// TIA Portal V18 export
// export: Created 2025-12-01T12:38:34.6445112Z, ExportSetting None, DisplayName Totally Integrated Automation Portal, DisplayVersion V18 Update 5, DisplayName TIA Portal Openness, DisplayVersion V18 Update 5, DisplayName TIA Portal Teamcenter Gateway, DisplayVersion V18, DisplayName TIA Portal Version Control Interface, DisplayVersion V18, DisplayName STEP 7 Professional, DisplayVersion V18 Update 5, DisplayName STEP 7 Safety, DisplayVersion V18, DisplayName WinCC Professional, DisplayVersion V18 Update 5
FUNCTION_BLOCK "ST10_Stopper_FB"   // FB1160, LAD
{ S7_Optimized_Access := 'TRUE' }
// stored: AutoNumber false, MemoryReserve 100, SetENOAutomatically false
   VAR
      FB_Stopper_Instance { S7_SetPoint := 'True'} : Array[1..3] of "FB_Stopper";
   END_VAR
BEGIN

REGION Network 1 (SCL): A-托盘缓存阻挡气缸
       (*  
       REGION 允许释放条件,根据实际完善
           //马达运行中且工位一允许进料
           IF "ST350_Motor_InterfaceDB".aDev[1].Run  THEN
               "ST350_Stopper_InterfaceDB".Command[1].In.iReleaseClear := TRUE;
           ELSE
               "ST350_Stopper_InterfaceDB".Command[1].In.iReleaseClear := FALSE;
           END_IF;
       END_REGION

       REGION IO_image
           //InPut
           "ST350_Stopper_InterfaceDB".Command[1].In.iSensor := "iBurfferPalletDetection";//本站托盘到位
           "ST350_Stopper_InterfaceDB".Command[1].In.iNextSensor := "iWork01PalletDetection";//后站托盘到位
           "ST350_Stopper_InterfaceDB".Command[1].In.iNextValve := "oA-Lifting-01StopperCylinder";//后站挡停输出

           // //OutPut
            "ST10Cylinder".Cy[5].Inout.AutoGoWork:= "ST350_Stopper_InterfaceDB".Command[1].Out.oValve;//本站挡停输出
       END_REGION


       *)
END_REGION

REGION Network 2: #FB_Stopper_Instance[1] A-托盘缓存阻挡气缸
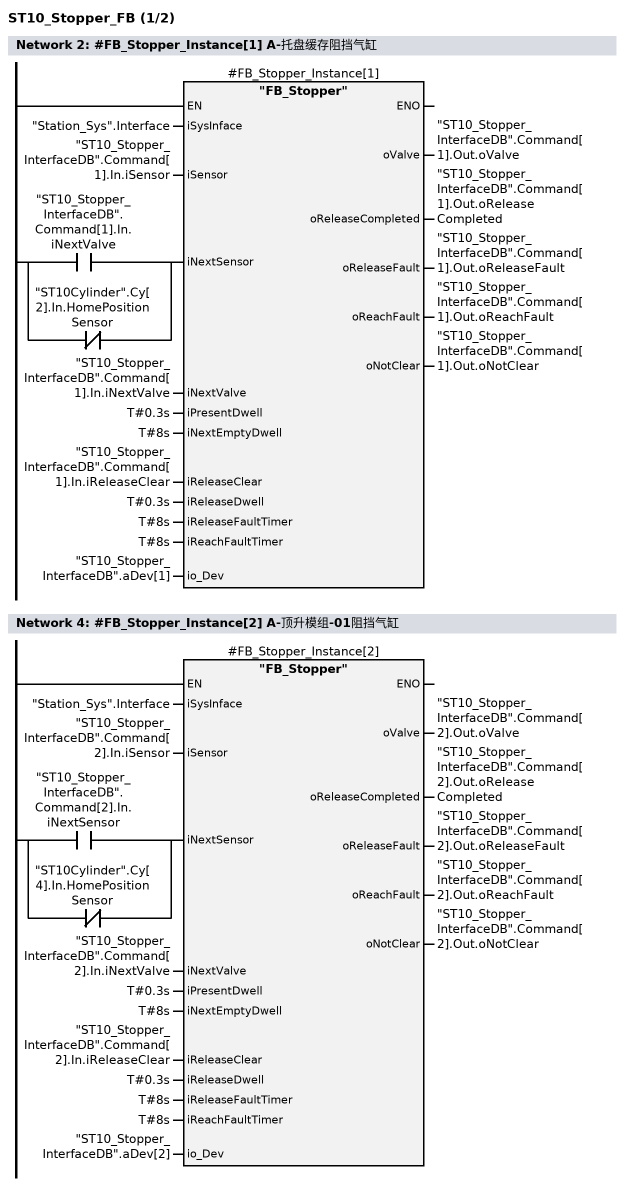
   RUNG wire#powerrail
      #FB_Stopper_Instance[1](iNextSensor := wire#w1, iSysInface := "Station_Sys".Interface, iSensor := "ST10_Stopper_InterfaceDB".Command[1].In.iSensor, iNextValve := "ST10_Stopper_InterfaceDB".Command[1].In.iNextValve, iPresentDwell := T#0.3s, iNextEmptyDwell := T#8s, iReleaseClear := "ST10_Stopper_InterfaceDB".Command[1].In.iReleaseClear, iReleaseDwell := T#0.3s, iReleaseFaultTimer := T#8s, iReachFaultTimer := T#8s, io_Dev := "ST10_Stopper_InterfaceDB".aDev[1], oValve => "ST10_Stopper_InterfaceDB".Command[1].Out.oValve, oReleaseCompleted => "ST10_Stopper_InterfaceDB".Command[1].Out.oReleaseCompleted, oReleaseFault => "ST10_Stopper_InterfaceDB".Command[1].Out.oReleaseFault, oReachFault => "ST10_Stopper_InterfaceDB".Command[1].Out.oReachFault, oNotClear => "ST10_Stopper_InterfaceDB".Command[1].Out.oNotClear)
   END_RUNG
   RUNG wire#powerrail
      Contact( "ST10_Stopper_InterfaceDB".Command[1].In.iNextValve )
   END_RUNG wire#w1
   RUNG wire#powerrail
      I_Contact( "ST10Cylinder".Cy[2].In.HomePositionSensor )
   END_RUNG wire#w1
   // the same network as SCL:
   #FB_Stopper_Instance[1](iSysInface := "Station_Sys".Interface,   // "FB_Stopper"
                           iSensor := "ST10_Stopper_InterfaceDB".Command[1].In.iSensor,
                           iNextSensor := "ST10_Stopper_InterfaceDB".Command[1].In.iNextValve OR NOT "ST10Cylinder".Cy[2].In.HomePositionSensor,
                           iNextValve := "ST10_Stopper_InterfaceDB".Command[1].In.iNextValve,
                           iPresentDwell := T#0.3s,
                           iNextEmptyDwell := T#8s,
                           iReleaseClear := "ST10_Stopper_InterfaceDB".Command[1].In.iReleaseClear,
                           iReleaseDwell := T#0.3s,
                           iReleaseFaultTimer := T#8s,
                           iReachFaultTimer := T#8s,
                           io_Dev := "ST10_Stopper_InterfaceDB".aDev[1],
                           oValve => "ST10_Stopper_InterfaceDB".Command[1].Out.oValve,
                           oReleaseCompleted => "ST10_Stopper_InterfaceDB".Command[1].Out.oReleaseCompleted,
                           oReleaseFault => "ST10_Stopper_InterfaceDB".Command[1].Out.oReleaseFault,
                           oReachFault => "ST10_Stopper_InterfaceDB".Command[1].Out.oReachFault,
                           oNotClear => "ST10_Stopper_InterfaceDB".Command[1].Out.oNotClear);
END_REGION

REGION Network 3 (SCL): A-顶升模组-01阻挡气缸
   (*
   REGION 允许释放条件,根据实际完善:顶升下降且线体运行中
       IF "ST10Cylinder".Cy[2].In.HomePositionSensor AND ("ST350_Motor_InterfaceDB".aDev[1].Run OR "Station_Sys".Manual.Mode) THEN//
           "ST350_Stopper_InterfaceDB".Command[2].In.iReleaseClear := True;
       ELSE
           "ST350_Stopper_InterfaceDB".Command[2].In.iReleaseClear := FALSE;
       END_IF;
   END_REGION

   REGION IO_image
       //InPut
       "ST350_Stopper_InterfaceDB".Command[2].In.iSensor := "iWork01PalletDetection";//本站托盘到位
       "ST350_Stopper_InterfaceDB".Command[2].In.iNextSensor := "iWork02PalletDetection";//后站托盘到位
       "ST350_Stopper_InterfaceDB".Command[2].In.iNextValve := "oA-Lifting-02StopperCylinder";//后站挡停输出

       // //OutPut
        "ST10Cylinder".Cy[1].Inout.AutoGoWork:= "ST350_Stopper_InterfaceDB".Command[2].Out.oValve;//本站挡停输出
   END_REGION

   *0
END_REGION

REGION Network 4: #FB_Stopper_Instance[2] A-顶升模组-01阻挡气缸
   RUNG wire#powerrail
      #FB_Stopper_Instance[2](iNextSensor := wire#w1, iSysInface := "Station_Sys".Interface, iSensor := "ST10_Stopper_InterfaceDB".Command[2].In.iSensor, iNextValve := "ST10_Stopper_InterfaceDB".Command[2].In.iNextValve, iPresentDwell := T#0.3s, iNextEmptyDwell := T#8s, iReleaseClear := "ST10_Stopper_InterfaceDB".Command[2].In.iReleaseClear, iReleaseDwell := T#0.3s, iReleaseFaultTimer := T#8s, iReachFaultTimer := T#8s, io_Dev := "ST10_Stopper_InterfaceDB".aDev[2], oValve => "ST10_Stopper_InterfaceDB".Command[2].Out.oValve, oReleaseCompleted => "ST10_Stopper_InterfaceDB".Command[2].Out.oReleaseCompleted, oReleaseFault => "ST10_Stopper_InterfaceDB".Command[2].Out.oReleaseFault, oReachFault => "ST10_Stopper_InterfaceDB".Command[2].Out.oReachFault, oNotClear => "ST10_Stopper_InterfaceDB".Command[2].Out.oNotClear)
   END_RUNG
   RUNG wire#powerrail
      Contact( "ST10_Stopper_InterfaceDB".Command[2].In.iNextSensor )
   END_RUNG wire#w1
   RUNG wire#powerrail
      I_Contact( "ST10Cylinder".Cy[4].In.HomePositionSensor )
   END_RUNG wire#w1
   // the same network as SCL:
   #FB_Stopper_Instance[2](iSysInface := "Station_Sys".Interface,   // "FB_Stopper"
                           iSensor := "ST10_Stopper_InterfaceDB".Command[2].In.iSensor,
                           iNextSensor := "ST10_Stopper_InterfaceDB".Command[2].In.iNextSensor OR NOT "ST10Cylinder".Cy[4].In.HomePositionSensor,
                           iNextValve := "ST10_Stopper_InterfaceDB".Command[2].In.iNextValve,
                           iPresentDwell := T#0.3s,
                           iNextEmptyDwell := T#8s,
                           iReleaseClear := "ST10_Stopper_InterfaceDB".Command[2].In.iReleaseClear,
                           iReleaseDwell := T#0.3s,
                           iReleaseFaultTimer := T#8s,
                           iReachFaultTimer := T#8s,
                           io_Dev := "ST10_Stopper_InterfaceDB".aDev[2],
                           oValve => "ST10_Stopper_InterfaceDB".Command[2].Out.oValve,
                           oReleaseCompleted => "ST10_Stopper_InterfaceDB".Command[2].Out.oReleaseCompleted,
                           oReleaseFault => "ST10_Stopper_InterfaceDB".Command[2].Out.oReleaseFault,
                           oReachFault => "ST10_Stopper_InterfaceDB".Command[2].Out.oReachFault,
                           oNotClear => "ST10_Stopper_InterfaceDB".Command[2].Out.oNotClear);
END_REGION

REGION Network 5 (SCL): A-顶升模组-02阻挡气缸
   //允许释放条件,根据实际完善:顶升下降且线体运行中
   (*

   REGION IOimage
       //InPut
       "ST350_Stopper_InterfaceDB".Command[3].In.iSensor := "iWork02PalletDetection";//本站托盘到位
       "ST350_Stopper_InterfaceDB".Command[3].In.iNextSensor := "iD-LiftingDetection" AND NOT "iD-LiftingINDetection" ;//后站托盘到位

       //替换后站挡停释放信号：升降机在下&顶升下&无料&允许金托盘
       // "ST350_Stopper_InterfaceDB".Command[3].In.iNextValve := ;//后站挡停输出

       // //OutPut
        "ST10Cylinder".Cy[3].Inout.AutoGoWork := "ST350_Stopper_InterfaceDB".Command[3].Out.oValve;//本站挡停输出


   END_REGION

   *)
END_REGION

REGION Network 6: #FB_Stopper_Instance[3] A-顶升模组-02阻挡气缸
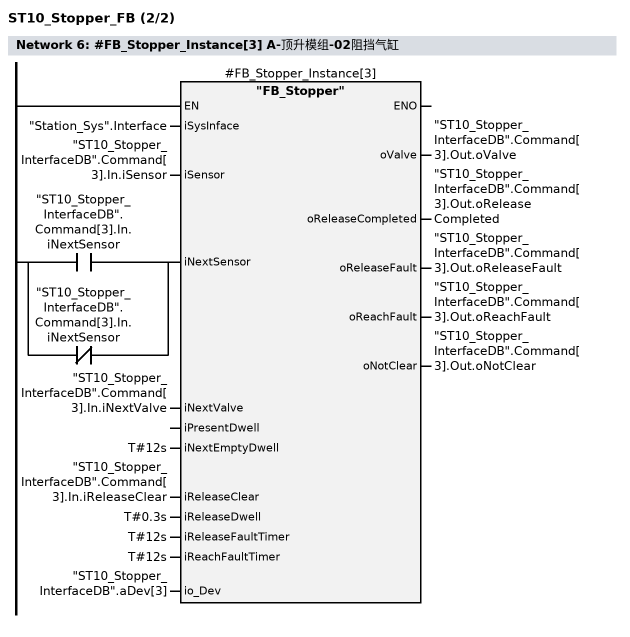
   RUNG wire#powerrail
      #FB_Stopper_Instance[3](iNextSensor := wire#w1, iSysInface := "Station_Sys".Interface, iSensor := "ST10_Stopper_InterfaceDB".Command[3].In.iSensor, iNextValve := "ST10_Stopper_InterfaceDB".Command[3].In.iNextValve, iPresentDwell :=, iNextEmptyDwell := T#12s, iReleaseClear := "ST10_Stopper_InterfaceDB".Command[3].In.iReleaseClear, iReleaseDwell := T#0.3s, iReleaseFaultTimer := T#12s, iReachFaultTimer := T#12s, io_Dev := "ST10_Stopper_InterfaceDB".aDev[3], oValve => "ST10_Stopper_InterfaceDB".Command[3].Out.oValve, oReleaseCompleted => "ST10_Stopper_InterfaceDB".Command[3].Out.oReleaseCompleted, oReleaseFault => "ST10_Stopper_InterfaceDB".Command[3].Out.oReleaseFault, oReachFault => "ST10_Stopper_InterfaceDB".Command[3].Out.oReachFault, oNotClear => "ST10_Stopper_InterfaceDB".Command[3].Out.oNotClear)
   END_RUNG
   RUNG wire#powerrail
      Contact( "ST10_Stopper_InterfaceDB".Command[3].In.iNextSensor )
   END_RUNG wire#w1
   RUNG wire#powerrail
      I_Contact( "ST10_Stopper_InterfaceDB".Command[3].In.iNextSensor )
   END_RUNG wire#w1
   // the same network as SCL:
   #FB_Stopper_Instance[3](iSysInface := "Station_Sys".Interface,   // "FB_Stopper"
                           iSensor := "ST10_Stopper_InterfaceDB".Command[3].In.iSensor,
                           iNextSensor := "ST10_Stopper_InterfaceDB".Command[3].In.iNextSensor OR NOT "ST10_Stopper_InterfaceDB".Command[3].In.iNextSensor,
                           iNextValve := "ST10_Stopper_InterfaceDB".Command[3].In.iNextValve,
                           iNextEmptyDwell := T#12s,
                           iReleaseClear := "ST10_Stopper_InterfaceDB".Command[3].In.iReleaseClear,
                           iReleaseDwell := T#0.3s,
                           iReleaseFaultTimer := T#12s,
                           iReachFaultTimer := T#12s,
                           io_Dev := "ST10_Stopper_InterfaceDB".aDev[3],
                           oValve => "ST10_Stopper_InterfaceDB".Command[3].Out.oValve,
                           oReleaseCompleted => "ST10_Stopper_InterfaceDB".Command[3].Out.oReleaseCompleted,
                           oReleaseFault => "ST10_Stopper_InterfaceDB".Command[3].Out.oReleaseFault,
                           oReachFault => "ST10_Stopper_InterfaceDB".Command[3].Out.oReachFault,
                           oNotClear => "ST10_Stopper_InterfaceDB".Command[3].Out.oNotClear);
END_REGION
END_FUNCTION_BLOCK
